// SIMATIC S7-200 project (STEP 7-Micro/WIN), CPU 224XP REL 02.00

ORGANIZATION_BLOCK 主程序:OB1
TITLE=程序注释
BEGIN
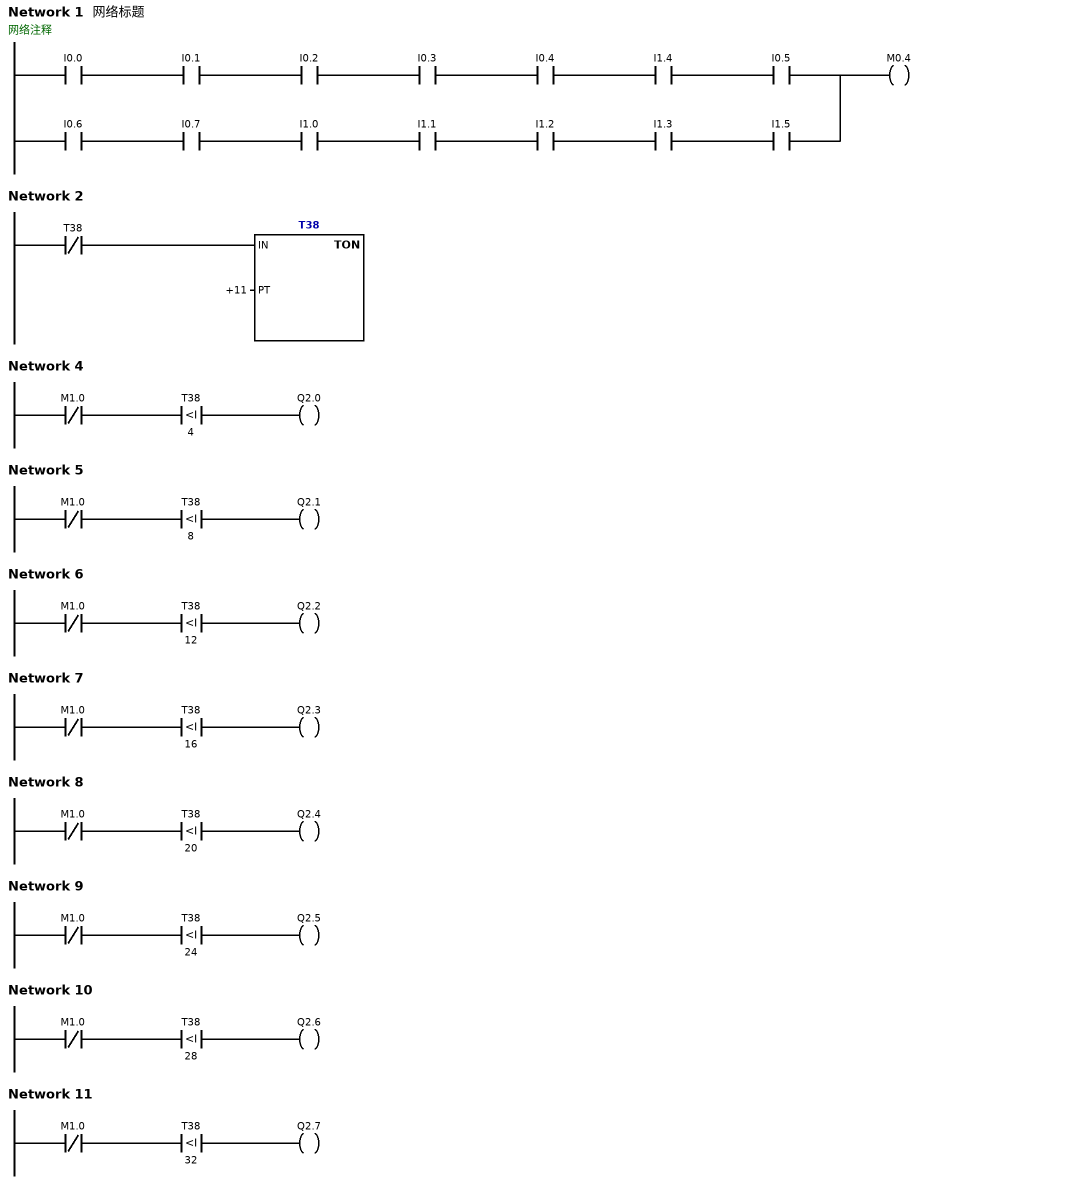
Network 1 // 网络标题
// 网络注释
// (network saved uncompiled; LAD cells follow)
// row 0: c0 -| |- I0.0  c1 -| |- I0.1  c2 -| |- I0.2  c3 -| |- I0.3  c4 -| |- I0.4  c5 -| |- I1.4  c6 -| |- I0.5 v  c7 -( ) M0.4
// row 1: c0 -| |- I0.6  c1 -| |- I0.7  c2 -| |- I1.0  c3 -| |- I1.1  c4 -| |- I1.2  c5 -| |- I1.3  c6 -| |- I1.5 ^
Network 2
// (network saved uncompiled; LAD cells follow)
// row 0: c0 -|/|- T38  c1 --  c2 [TON T38 IN:=power@row0, PT:=+11]
// row 1: c2 [box]
Network 4
// (network saved uncompiled; LAD cells follow)
// row 0: c0 -|/|- M1.0  c1 -|<I|- T38, 4  c2 -( ) Q2.0
Network 5
// (network saved uncompiled; LAD cells follow)
// row 0: c0 -|/|- M1.0  c1 -|<I|- T38, 8  c2 -( ) Q2.1
Network 6
// (network saved uncompiled; LAD cells follow)
// row 0: c0 -|/|- M1.0  c1 -|<I|- T38, 12  c2 -( ) Q2.2
Network 7
// (network saved uncompiled; LAD cells follow)
// row 0: c0 -|/|- M1.0  c1 -|<I|- T38, 16  c2 -( ) Q2.3
Network 8
// (network saved uncompiled; LAD cells follow)
// row 0: c0 -|/|- M1.0  c1 -|<I|- T38, 20  c2 -( ) Q2.4
Network 9
// (network saved uncompiled; LAD cells follow)
// row 0: c0 -|/|- M1.0  c1 -|<I|- T38, 24  c2 -( ) Q2.5
Network 10
// (network saved uncompiled; LAD cells follow)
// row 0: c0 -|/|- M1.0  c1 -|<I|- T38, 28  c2 -( ) Q2.6
Network 11
// (network saved uncompiled; LAD cells follow)
// row 0: c0 -|/|- M1.0  c1 -|<I|- T38, 32  c2 -( ) Q2.7
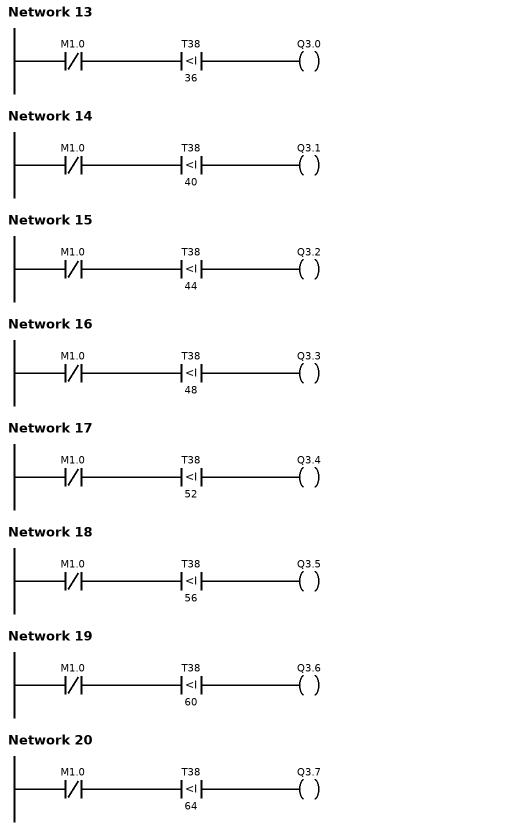
Network 13
// (network saved uncompiled; LAD cells follow)
// row 0: c0 -|/|- M1.0  c1 -|<I|- T38, 36  c2 -( ) Q3.0
Network 14
// (network saved uncompiled; LAD cells follow)
// row 0: c0 -|/|- M1.0  c1 -|<I|- T38, 40  c2 -( ) Q3.1
Network 15
// (network saved uncompiled; LAD cells follow)
// row 0: c0 -|/|- M1.0  c1 -|<I|- T38, 44  c2 -( ) Q3.2
Network 16
// (network saved uncompiled; LAD cells follow)
// row 0: c0 -|/|- M1.0  c1 -|<I|- T38, 48  c2 -( ) Q3.3
Network 17
// (network saved uncompiled; LAD cells follow)
// row 0: c0 -|/|- M1.0  c1 -|<I|- T38, 52  c2 -( ) Q3.4
Network 18
// (network saved uncompiled; LAD cells follow)
// row 0: c0 -|/|- M1.0  c1 -|<I|- T38, 56  c2 -( ) Q3.5
Network 19
// (network saved uncompiled; LAD cells follow)
// row 0: c0 -|/|- M1.0  c1 -|<I|- T38, 60  c2 -( ) Q3.6
Network 20
// (network saved uncompiled; LAD cells follow)
// row 0: c0 -|/|- M1.0  c1 -|<I|- T38, 64  c2 -( ) Q3.7
END_ORGANIZATION_BLOCK
